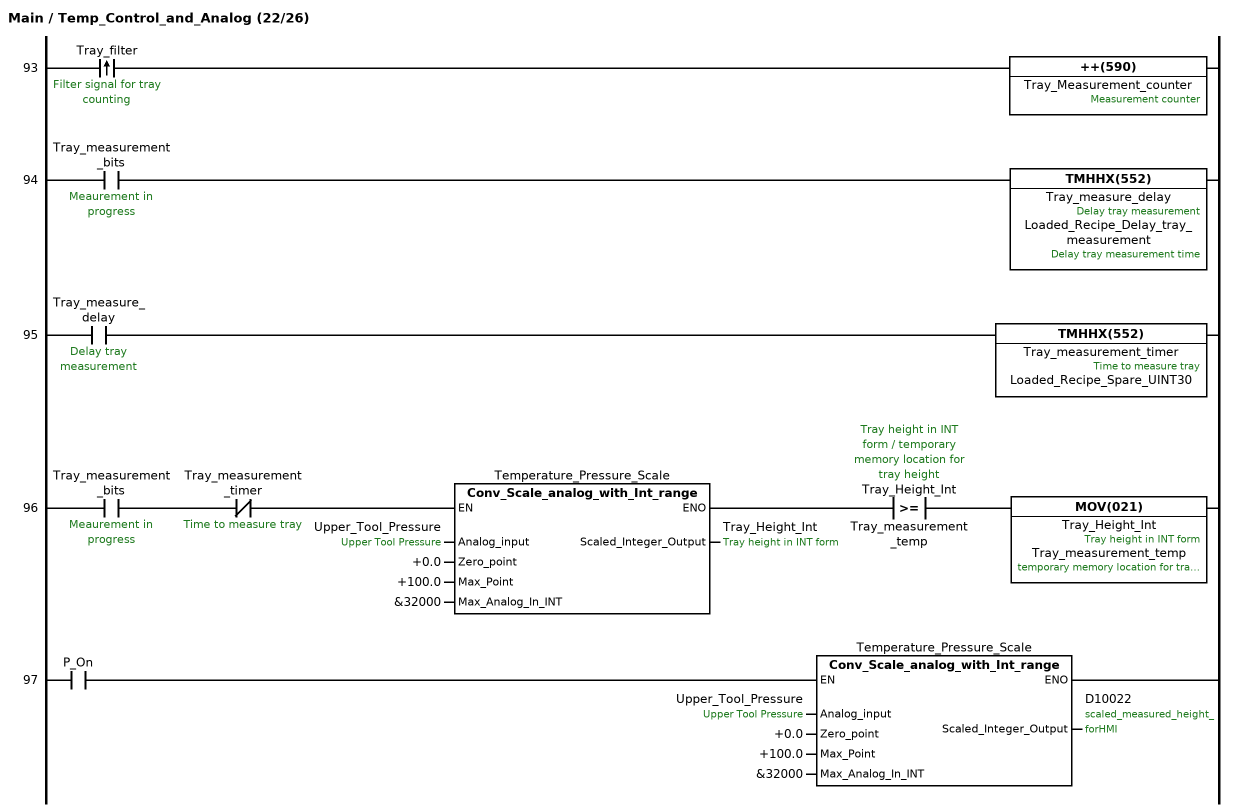
; [picture p120: Main / Temp_Control_and_Analog, rungs 93-97]
; rung 93
@LD Tray_filter  ; Filter signal for tray counting
++(590) Tray_Measurement_counter  ; Measurement counter
; rung 94
LD Tray_measurement_bits  ; Meaurement in progress
TMHHX(552) Tray_measure_delay Loaded_Recipe_Delay_tray_measurement  ; Delay tray measurement, Delay tray measurement time
; rung 95
LD Tray_measure_delay  ; Delay tray measurement
TMHHX(552) Tray_measurement_timer Loaded_Recipe_Spare_UINT30  ; Time to measure tray
; rung 96
LD Tray_measurement_bits  ; Meaurement in progress
ANDNOT Tray_measurement_timer  ; Time to measure tray
CALL Temperature_Pressure_Scale : Conv_Scale_analog_with_Int_range (Analog_input := Upper_Tool_Pressure, Zero_point := +0.0, Max_Point := +100.0, Max_Analog_In_INT := &32000, Scaled_Integer_Output => Tray_Height_Int)  ; Upper Tool Pressure, Tray height in INT form
AND>=(325) Tray_Height_Int Tray_measurement_temp  ; Tray height in INT form, temporary memory location for tray height
MOV(021) Tray_Height_Int Tray_measurement_temp  ; Tray height in INT form, temporary memory location for tray height
; rung 97
LD P_On
CALL Temperature_Pressure_Scale : Conv_Scale_analog_with_Int_range (Analog_input := Upper_Tool_Pressure, Zero_point := +0.0, Max_Point := +100.0, Max_Analog_In_INT := &32000, Scaled_Integer_Output => D10022)  ; Upper Tool Pressure, scaled_measured_height_forHMI

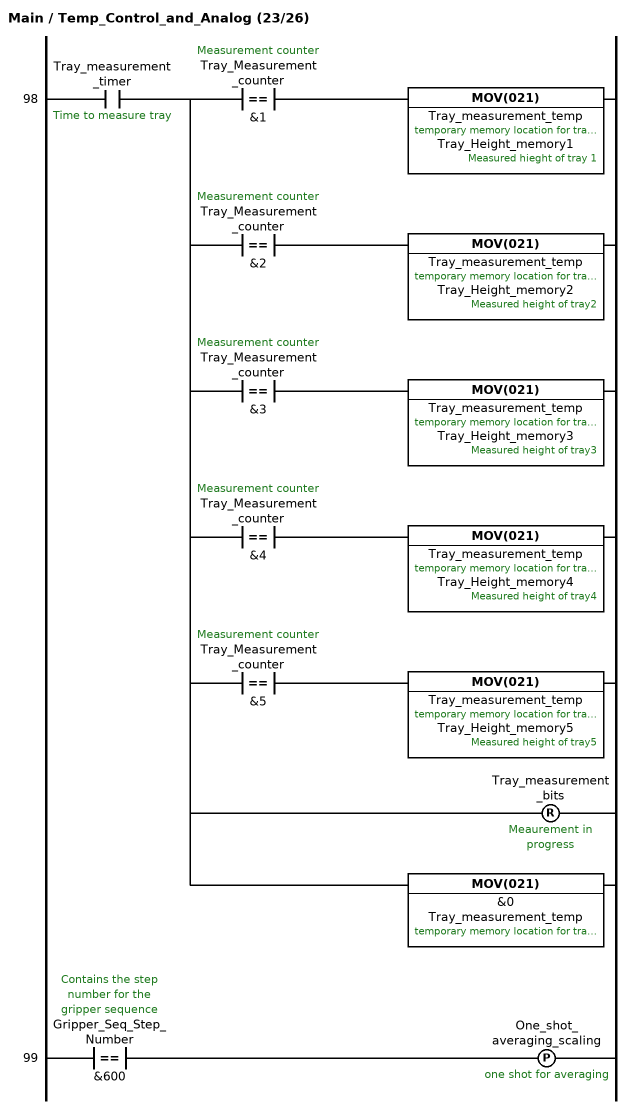
; rung 98
LD Tray_measurement_timer  ; Time to measure tray
OUT TR0
AND=(300) Tray_Measurement_counter &1  ; Measurement counter
MOV(021) Tray_measurement_temp Tray_Height_memory1  ; temporary memory location for tray height, Measured hieght of tray 1
LD TR0
AND=(300) Tray_Measurement_counter &2  ; Measurement counter
MOV(021) Tray_measurement_temp Tray_Height_memory2  ; temporary memory location for tray height, Measured height of tray2
LD TR0
AND=(300) Tray_Measurement_counter &3  ; Measurement counter
MOV(021) Tray_measurement_temp Tray_Height_memory3  ; temporary memory location for tray height, Measured height of tray3
LD TR0
AND=(300) Tray_Measurement_counter &4  ; Measurement counter
MOV(021) Tray_measurement_temp Tray_Height_memory4  ; temporary memory location for tray height, Measured height of tray4
LD TR0
AND=(300) Tray_Measurement_counter &5  ; Measurement counter
MOV(021) Tray_measurement_temp Tray_Height_memory5  ; temporary memory location for tray height, Measured height of tray5
LD TR0
RSET Tray_measurement_bits  ; Meaurement in progress
MOV(021) &0 Tray_measurement_temp  ; temporary memory location for tray height
; rung 99
LD=(300) Gripper_Seq_Step_Number &600  ; Contains the step number for the gripper sequence
DIFU(013) One_shot_averaging_scaling  ; one shot for averaging

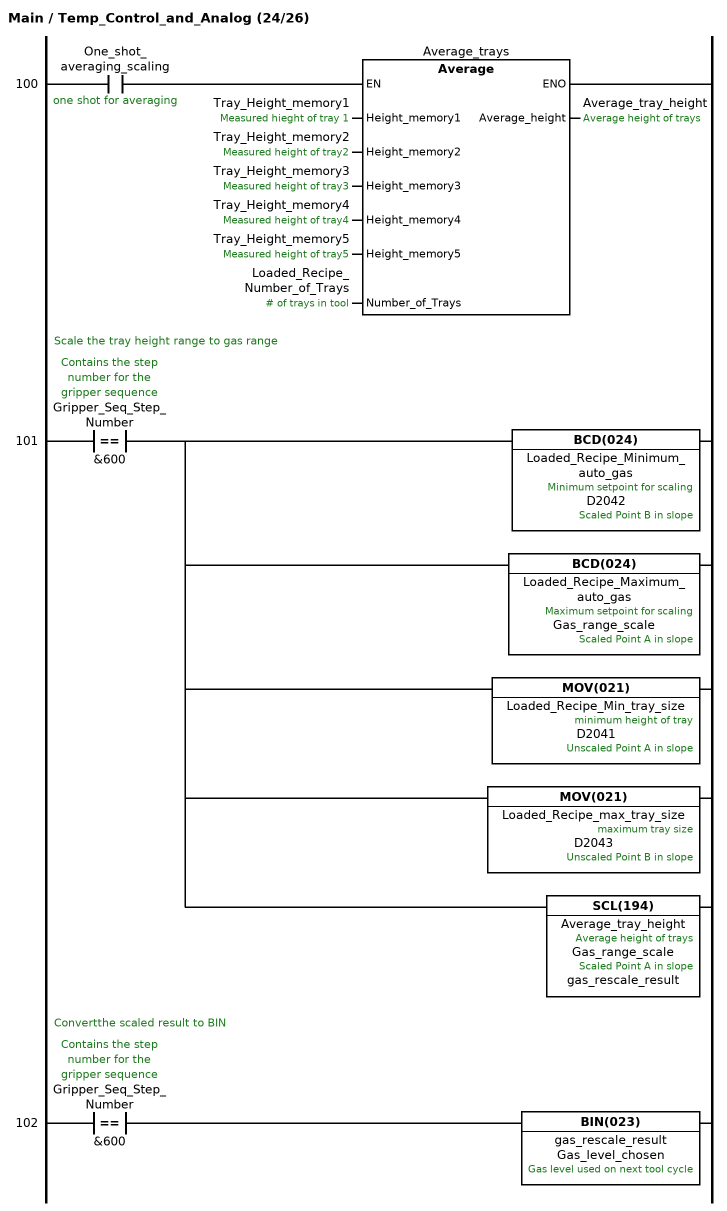
; rung 100
LD One_shot_averaging_scaling  ; one shot for averaging
CALL Average_trays : Average (Height_memory1 := Tray_Height_memory1, Height_memory2 := Tray_Height_memory2, Height_memory3 := Tray_Height_memory3, Height_memory4 := Tray_Height_memory4, Height_memory5 := Tray_Height_memory5, Number_of_Trays := Loaded_Recipe_Number_of_Trays, Average_height => Average_tray_height)  ; Measured hieght of tray 1, Measured height of tray2, Measured height of tray3, Measured height of tray4, Measured height of tray5, # of trays in tool, Average height of trays
; rung 101: Scale the tray height range to gas range
LD=(300) Gripper_Seq_Step_Number &600  ; Contains the step number for the gripper sequence
BCD(024) Loaded_Recipe_Minimum_auto_gas D2042  ; Minimum setpoint for scaling, Scaled Point B in slope
BCD(024) Loaded_Recipe_Maximum_auto_gas Gas_range_scale  ; Maximum setpoint for scaling, Scaled Point A in slope
MOV(021) Loaded_Recipe_Min_tray_size D2041  ; minimum height of tray, Unscaled Point A in slope
MOV(021) Loaded_Recipe_max_tray_size D2043  ; maximum tray size, Unscaled Point B in slope
SCL(194) Average_tray_height Gas_range_scale gas_rescale_result  ; Average height of trays, Scaled Point A in slope
; rung 102: Convertthe scaled result to BIN
LD=(300) Gripper_Seq_Step_Number &600  ; Contains the step number for the gripper sequence
BIN(023) gas_rescale_result Gas_level_chosen  ; Gas level used on next tool cycle

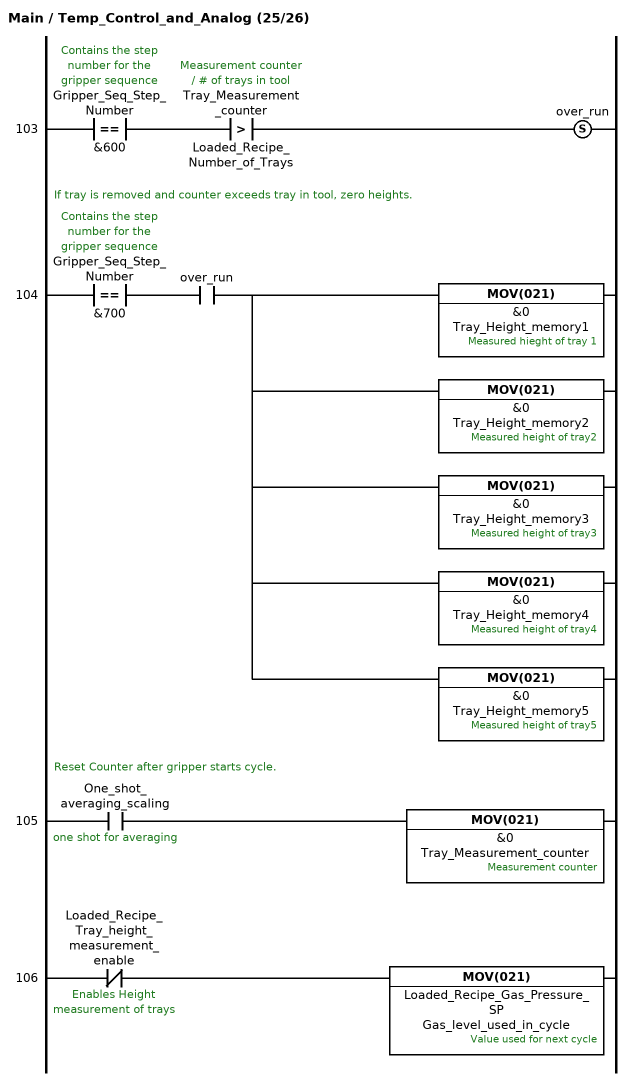
; rung 103
LD=(300) Gripper_Seq_Step_Number &600  ; Contains the step number for the gripper sequence
AND>(320) Tray_Measurement_counter Loaded_Recipe_Number_of_Trays  ; Measurement counter, # of trays in tool
SET over_run
; rung 104: If tray is removed and counter exceeds tray in tool, zero heights.
LD=(300) Gripper_Seq_Step_Number &700  ; Contains the step number for the gripper sequence
AND over_run
MOV(021) &0 Tray_Height_memory1  ; Measured hieght of tray 1
MOV(021) &0 Tray_Height_memory2  ; Measured height of tray2
MOV(021) &0 Tray_Height_memory3  ; Measured height of tray3
MOV(021) &0 Tray_Height_memory4  ; Measured height of tray4
MOV(021) &0 Tray_Height_memory5  ; Measured height of tray5
; rung 105: Reset Counter after gripper starts cycle.
LD One_shot_averaging_scaling  ; one shot for averaging
MOV(021) &0 Tray_Measurement_counter  ; Measurement counter
; rung 106
LDNOT Loaded_Recipe_Tray_height_measurement_enable  ; Enables Height measurement of trays
MOV(021) Loaded_Recipe_Gas_Pressure_SP Gas_level_used_in_cycle  ; Value used for next cycle

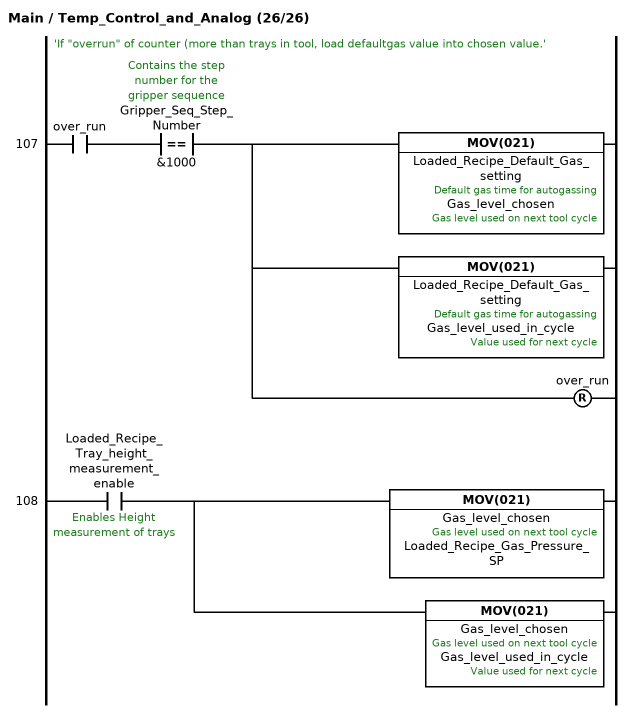
; rung 107: 'If "overrun" of counter (more than trays in tool, load defaultgas value into chosen value.'
LD over_run
AND=(300) Gripper_Seq_Step_Number &1000  ; Contains the step number for the gripper sequence
MOV(021) Loaded_Recipe_Default_Gas_setting Gas_level_chosen  ; Default gas time for autogassing, Gas level used on next tool cycle
MOV(021) Loaded_Recipe_Default_Gas_setting Gas_level_used_in_cycle  ; Default gas time for autogassing, Value used for next cycle
RSET over_run
; rung 108
LD Loaded_Recipe_Tray_height_measurement_enable  ; Enables Height measurement of trays
MOV(021) Gas_level_chosen Loaded_Recipe_Gas_Pressure_SP  ; Gas level used on next tool cycle
MOV(021) Gas_level_chosen Gas_level_used_in_cycle  ; Gas level used on next tool cycle, Value used for next cycle

### Section IOHandling

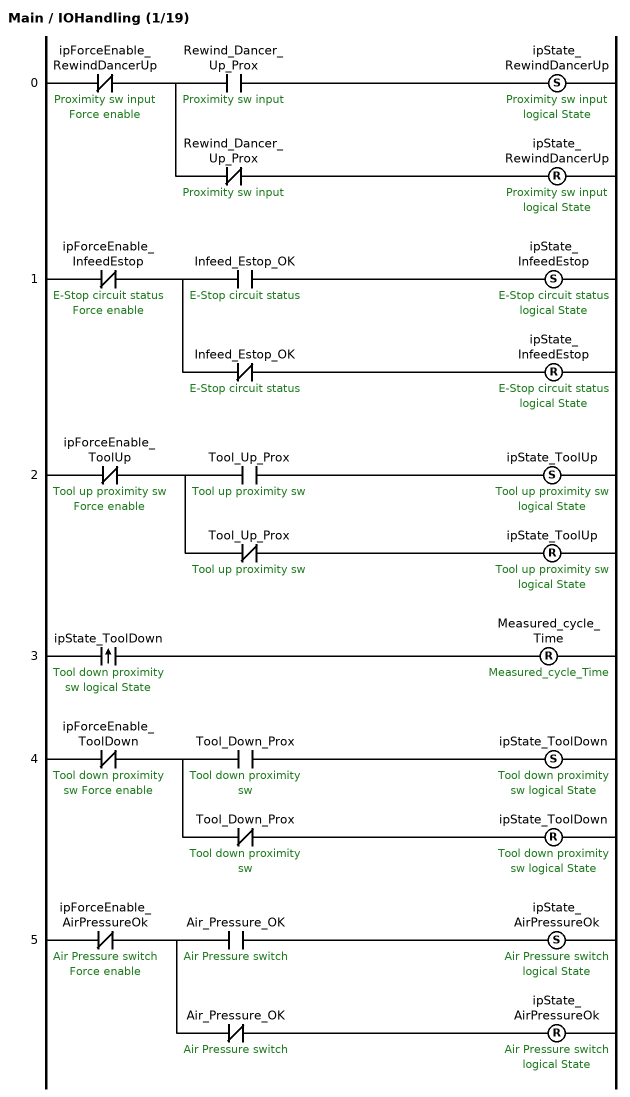
; rung 0
LDNOT ipForceEnable_RewindDancerUp  ; Proximity sw input Force enable
OUT TR0
AND Rewind_Dancer_Up_Prox  ; Proximity sw input
SET ipState_RewindDancerUp  ; Proximity sw input logical State
LD TR0
ANDNOT Rewind_Dancer_Up_Prox  ; Proximity sw input
RSET ipState_RewindDancerUp  ; Proximity sw input logical State
; rung 1
LDNOT ipForceEnable_InfeedEstop  ; E-Stop circuit status Force enable
OUT TR0
AND Infeed_Estop_OK  ; E-Stop circuit status
SET ipState_InfeedEstop  ; E-Stop circuit status logical State
LD TR0
ANDNOT Infeed_Estop_OK  ; E-Stop circuit status
RSET ipState_InfeedEstop  ; E-Stop circuit status logical State
; rung 2
LDNOT ipForceEnable_ToolUp  ; Tool up proximity sw Force enable
OUT TR0
AND Tool_Up_Prox  ; Tool up proximity sw
SET ipState_ToolUp  ; Tool up proximity sw logical State
LD TR0
ANDNOT Tool_Up_Prox  ; Tool up proximity sw
RSET ipState_ToolUp  ; Tool up proximity sw logical State
; rung 3
@LD ipState_ToolDown  ; Tool down proximity sw logical State
RSET Measured_cycle_Time  ; Measured_cycle_Time
; rung 4
LDNOT ipForceEnable_ToolDown  ; Tool down proximity sw Force enable
OUT TR0
AND Tool_Down_Prox  ; Tool down proximity sw
SET ipState_ToolDown  ; Tool down proximity sw logical State
LD TR0
ANDNOT Tool_Down_Prox  ; Tool down proximity sw
RSET ipState_ToolDown  ; Tool down proximity sw logical State
; rung 5
LDNOT ipForceEnable_AirPressureOk  ; Air Pressure switch Force enable
OUT TR0
AND Air_Pressure_OK  ; Air Pressure switch
SET ipState_AirPressureOk  ; Air Pressure switch logical State
LD TR0
ANDNOT Air_Pressure_OK  ; Air Pressure switch
RSET ipState_AirPressureOk  ; Air Pressure switch logical State

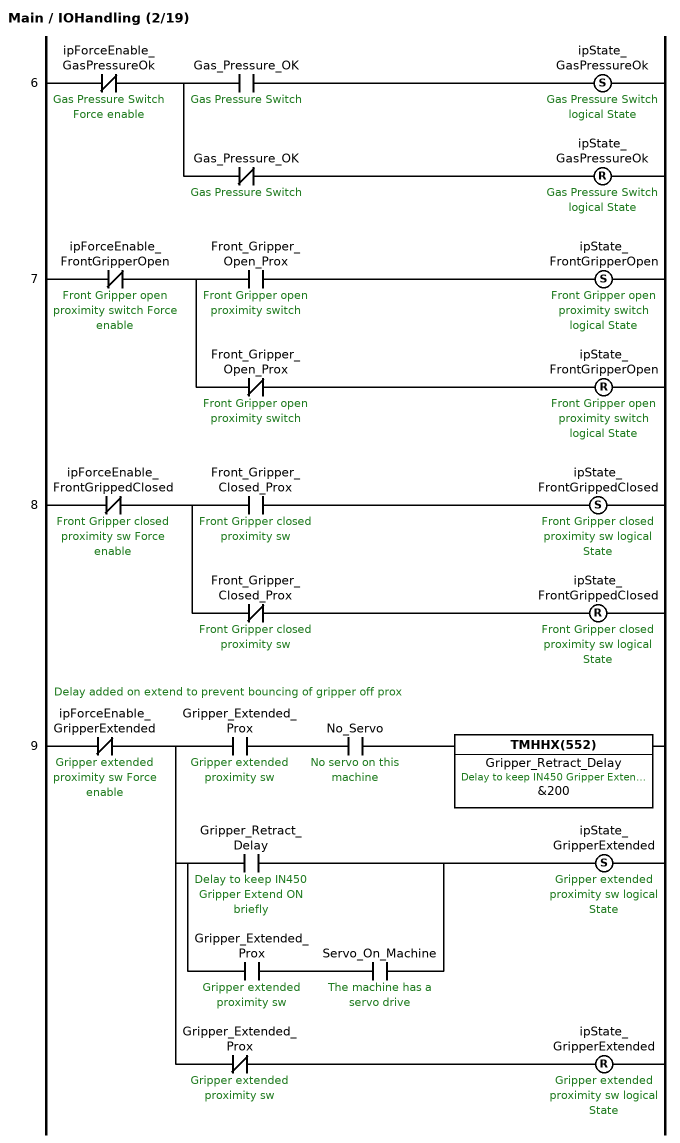
; rung 6
LDNOT ipForceEnable_GasPressureOk  ; Gas Pressure Switch Force enable
OUT TR0
AND Gas_Pressure_OK  ; Gas Pressure Switch
SET ipState_GasPressureOk  ; Gas Pressure Switch logical State
LD TR0
ANDNOT Gas_Pressure_OK  ; Gas Pressure Switch
RSET ipState_GasPressureOk  ; Gas Pressure Switch logical State
; rung 7
LDNOT ipForceEnable_FrontGripperOpen  ; Front Gripper open proximity switch Force enable
OUT TR0
AND Front_Gripper_Open_Prox  ; Front Gripper open proximity switch
SET ipState_FrontGripperOpen  ; Front Gripper open proximity switch logical State
LD TR0
ANDNOT Front_Gripper_Open_Prox  ; Front Gripper open proximity switch
RSET ipState_FrontGripperOpen  ; Front Gripper open proximity switch logical State
; rung 8
LDNOT ipForceEnable_FrontGrippedClosed  ; Front Gripper closed proximity sw Force enable
OUT TR0
AND Front_Gripper_Closed_Prox  ; Front Gripper closed proximity sw
SET ipState_FrontGrippedClosed  ; Front Gripper closed proximity sw logical State
LD TR0
ANDNOT Front_Gripper_Closed_Prox  ; Front Gripper closed proximity sw
RSET ipState_FrontGrippedClosed  ; Front Gripper closed proximity sw logical State
; rung 9: Delay added on extend to prevent bouncing of gripper off prox
LDNOT ipForceEnable_GripperExtended  ; Gripper extended proximity sw Force enable
OUT TR0
AND Gripper_Extended_Prox  ; Gripper extended proximity sw
AND No_Servo  ; No servo on this machine
TMHHX(552) Gripper_Retract_Delay &200  ; Delay to keep IN450 Gripper Extend ON briefly
LD TR0
LD Gripper_Retract_Delay  ; Delay to keep IN450 Gripper Extend ON briefly
LD Gripper_Extended_Prox  ; Gripper extended proximity sw
AND Servo_On_Machine  ; The machine has a servo drive
ORLD
ANDLD
SET ipState_GripperExtended  ; Gripper extended proximity sw logical State
LD TR0
ANDNOT Gripper_Extended_Prox  ; Gripper extended proximity sw
RSET ipState_GripperExtended  ; Gripper extended proximity sw logical State

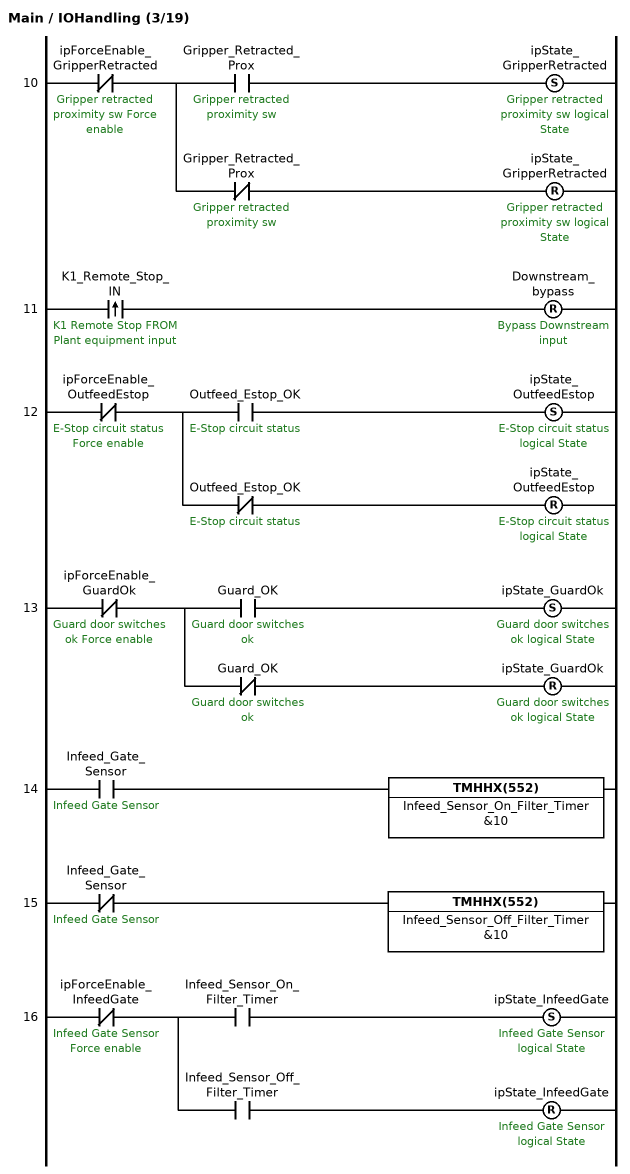
; rung 10
LDNOT ipForceEnable_GripperRetracted  ; Gripper retracted proximity sw Force enable
OUT TR0
AND Gripper_Retracted_Prox  ; Gripper retracted proximity sw
SET ipState_GripperRetracted  ; Gripper retracted proximity sw logical State
LD TR0
ANDNOT Gripper_Retracted_Prox  ; Gripper retracted proximity sw
RSET ipState_GripperRetracted  ; Gripper retracted proximity sw logical State
; rung 11
@LD K1_Remote_Stop_IN  ; K1 Remote Stop FROM Plant equipment input
RSET Downstream_bypass  ; Bypass Downstream input
; rung 12
LDNOT ipForceEnable_OutfeedEstop  ; E-Stop circuit status Force enable
OUT TR0
AND Outfeed_Estop_OK  ; E-Stop circuit status
SET ipState_OutfeedEstop  ; E-Stop circuit status logical State
LD TR0
ANDNOT Outfeed_Estop_OK  ; E-Stop circuit status
RSET ipState_OutfeedEstop  ; E-Stop circuit status logical State
; rung 13
LDNOT ipForceEnable_GuardOk  ; Guard door switches ok Force enable
OUT TR0
AND Guard_OK  ; Guard door switches ok
SET ipState_GuardOk  ; Guard door switches ok logical State
LD TR0
ANDNOT Guard_OK  ; Guard door switches ok
RSET ipState_GuardOk  ; Guard door switches ok logical State
; rung 14
LD Infeed_Gate_Sensor  ; Infeed Gate Sensor
TMHHX(552) Infeed_Sensor_On_Filter_Timer &10
; rung 15
LDNOT Infeed_Gate_Sensor  ; Infeed Gate Sensor
TMHHX(552) Infeed_Sensor_Off_Filter_Timer &10
; rung 16
LDNOT ipForceEnable_InfeedGate  ; Infeed Gate Sensor Force enable
OUT TR0
AND Infeed_Sensor_On_Filter_Timer
SET ipState_InfeedGate  ; Infeed Gate Sensor logical State
LD TR0
AND Infeed_Sensor_Off_Filter_Timer
RSET ipState_InfeedGate  ; Infeed Gate Sensor logical State

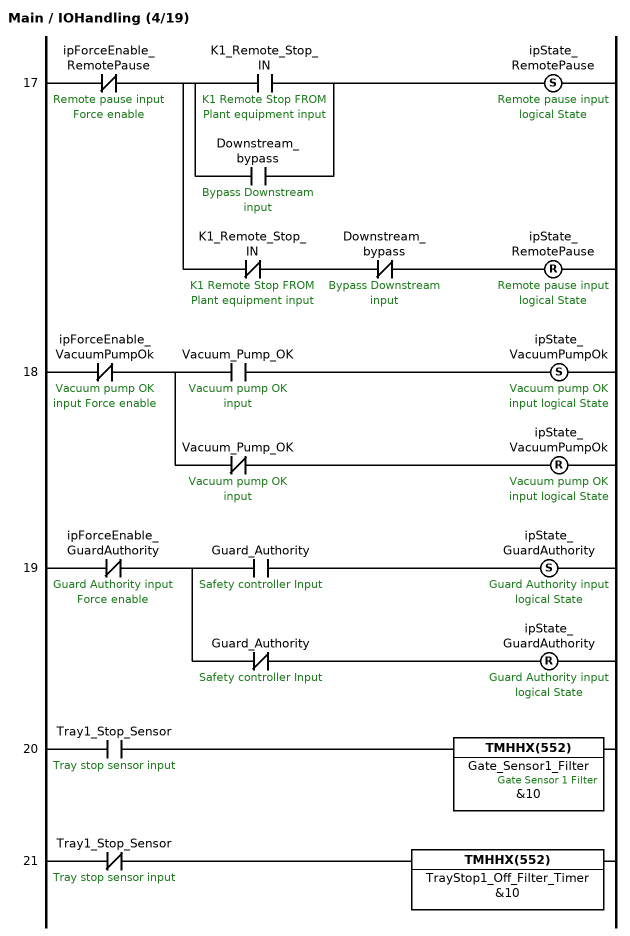
; rung 17
LDNOT ipForceEnable_RemotePause  ; Remote pause input Force enable
OUT TR0
LD K1_Remote_Stop_IN  ; K1 Remote Stop FROM Plant equipment input
OR Downstream_bypass  ; Bypass Downstream input
ANDLD
SET ipState_RemotePause  ; Remote pause input logical State
LD TR0
ANDNOT K1_Remote_Stop_IN  ; K1 Remote Stop FROM Plant equipment input
ANDNOT Downstream_bypass  ; Bypass Downstream input
RSET ipState_RemotePause  ; Remote pause input logical State
; rung 18
LDNOT ipForceEnable_VacuumPumpOk  ; Vacuum pump OK input Force enable
OUT TR0
AND Vacuum_Pump_OK  ; Vacuum pump OK input
SET ipState_VacuumPumpOk  ; Vacuum pump OK input logical State
LD TR0
ANDNOT Vacuum_Pump_OK  ; Vacuum pump OK input
RSET ipState_VacuumPumpOk  ; Vacuum pump OK input logical State
; rung 19
LDNOT ipForceEnable_GuardAuthority  ; Guard Authority input Force enable
OUT TR0
AND Guard_Authority  ; Safety controller Input
SET ipState_GuardAuthority  ; Guard Authority input logical State
LD TR0
ANDNOT Guard_Authority  ; Safety controller Input
RSET ipState_GuardAuthority  ; Guard Authority input logical State
; rung 20
LD Tray1_Stop_Sensor  ; Tray stop sensor input
TMHHX(552) Gate_Sensor1_Filter &10  ; Gate Sensor 1 Filter
; rung 21
LDNOT Tray1_Stop_Sensor  ; Tray stop sensor input
TMHHX(552) TrayStop1_Off_Filter_Timer &10

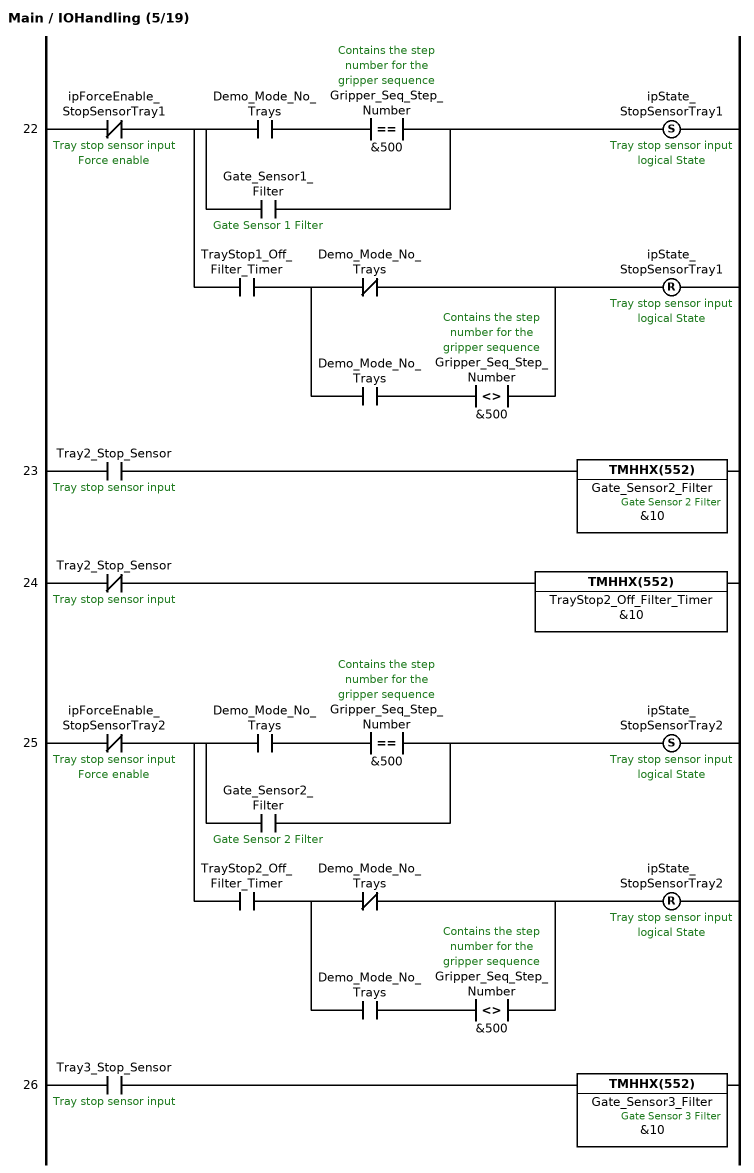
; rung 22
LDNOT ipForceEnable_StopSensorTray1  ; Tray stop sensor input Force enable
OUT TR0
LD Demo_Mode_No_Trays
AND=(300) Gripper_Seq_Step_Number &500  ; Contains the step number for the gripper sequence
OR Gate_Sensor1_Filter  ; Gate Sensor 1 Filter
ANDLD
SET ipState_StopSensorTray1  ; Tray stop sensor input logical State
LD TR0
AND TrayStop1_Off_Filter_Timer
LDNOT Demo_Mode_No_Trays
LD Demo_Mode_No_Trays
AND<>(305) Gripper_Seq_Step_Number &500  ; Contains the step number for the gripper sequence
ORLD
ANDLD
RSET ipState_StopSensorTray1  ; Tray stop sensor input logical State
; rung 23
LD Tray2_Stop_Sensor  ; Tray stop sensor input
TMHHX(552) Gate_Sensor2_Filter &10  ; Gate Sensor 2 Filter
; rung 24
LDNOT Tray2_Stop_Sensor  ; Tray stop sensor input
TMHHX(552) TrayStop2_Off_Filter_Timer &10
; rung 25
LDNOT ipForceEnable_StopSensorTray2  ; Tray stop sensor input Force enable
OUT TR0
LD Demo_Mode_No_Trays
AND=(300) Gripper_Seq_Step_Number &500  ; Contains the step number for the gripper sequence
OR Gate_Sensor2_Filter  ; Gate Sensor 2 Filter
ANDLD
SET ipState_StopSensorTray2  ; Tray stop sensor input logical State
LD TR0
AND TrayStop2_Off_Filter_Timer
LDNOT Demo_Mode_No_Trays
LD Demo_Mode_No_Trays
AND<>(305) Gripper_Seq_Step_Number &500  ; Contains the step number for the gripper sequence
ORLD
ANDLD
RSET ipState_StopSensorTray2  ; Tray stop sensor input logical State
; rung 26
LD Tray3_Stop_Sensor  ; Tray stop sensor input
TMHHX(552) Gate_Sensor3_Filter &10  ; Gate Sensor 3 Filter

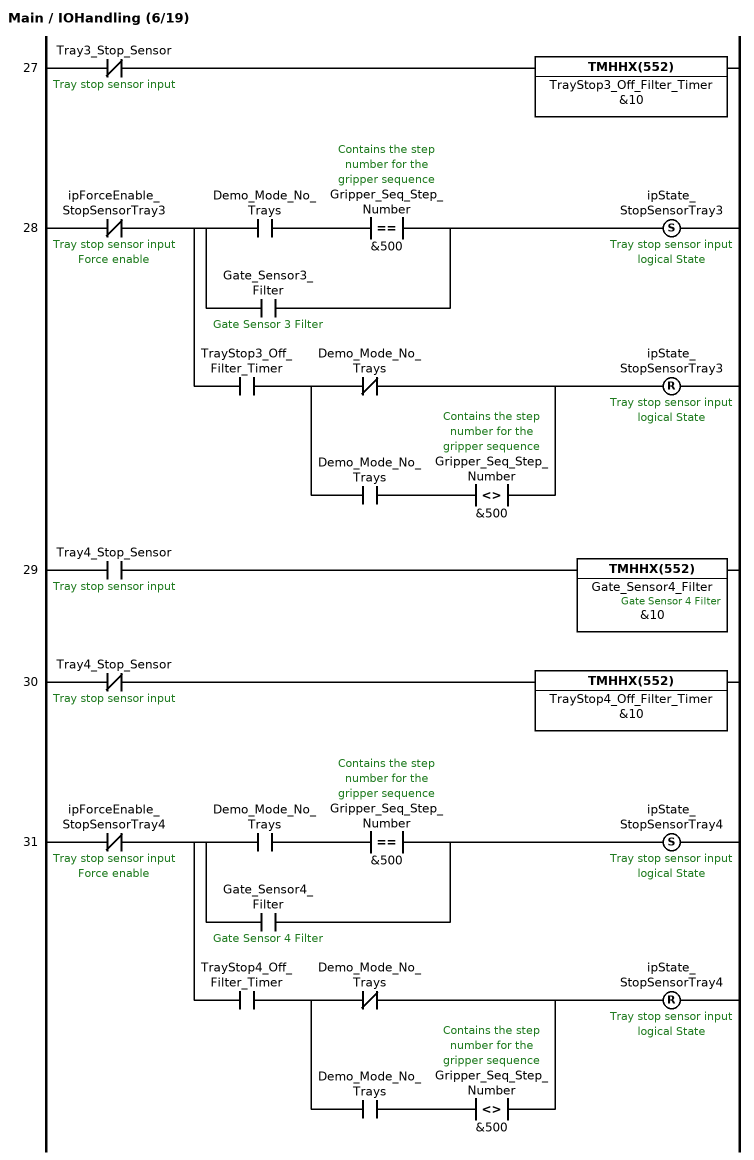
; rung 27
LDNOT Tray3_Stop_Sensor  ; Tray stop sensor input
TMHHX(552) TrayStop3_Off_Filter_Timer &10
; rung 28
LDNOT ipForceEnable_StopSensorTray3  ; Tray stop sensor input Force enable
OUT TR0
LD Demo_Mode_No_Trays
AND=(300) Gripper_Seq_Step_Number &500  ; Contains the step number for the gripper sequence
OR Gate_Sensor3_Filter  ; Gate Sensor 3 Filter
ANDLD
SET ipState_StopSensorTray3  ; Tray stop sensor input logical State
LD TR0
AND TrayStop3_Off_Filter_Timer
LDNOT Demo_Mode_No_Trays
LD Demo_Mode_No_Trays
AND<>(305) Gripper_Seq_Step_Number &500  ; Contains the step number for the gripper sequence
ORLD
ANDLD
RSET ipState_StopSensorTray3  ; Tray stop sensor input logical State
; rung 29
LD Tray4_Stop_Sensor  ; Tray stop sensor input
TMHHX(552) Gate_Sensor4_Filter &10  ; Gate Sensor 4 Filter
; rung 30
LDNOT Tray4_Stop_Sensor  ; Tray stop sensor input
TMHHX(552) TrayStop4_Off_Filter_Timer &10
; rung 31
LDNOT ipForceEnable_StopSensorTray4  ; Tray stop sensor input Force enable
OUT TR0
LD Demo_Mode_No_Trays
AND=(300) Gripper_Seq_Step_Number &500  ; Contains the step number for the gripper sequence
OR Gate_Sensor4_Filter  ; Gate Sensor 4 Filter
ANDLD
SET ipState_StopSensorTray4  ; Tray stop sensor input logical State
LD TR0
AND TrayStop4_Off_Filter_Timer
LDNOT Demo_Mode_No_Trays
LD Demo_Mode_No_Trays
AND<>(305) Gripper_Seq_Step_Number &500  ; Contains the step number for the gripper sequence
ORLD
ANDLD
RSET ipState_StopSensorTray4  ; Tray stop sensor input logical State

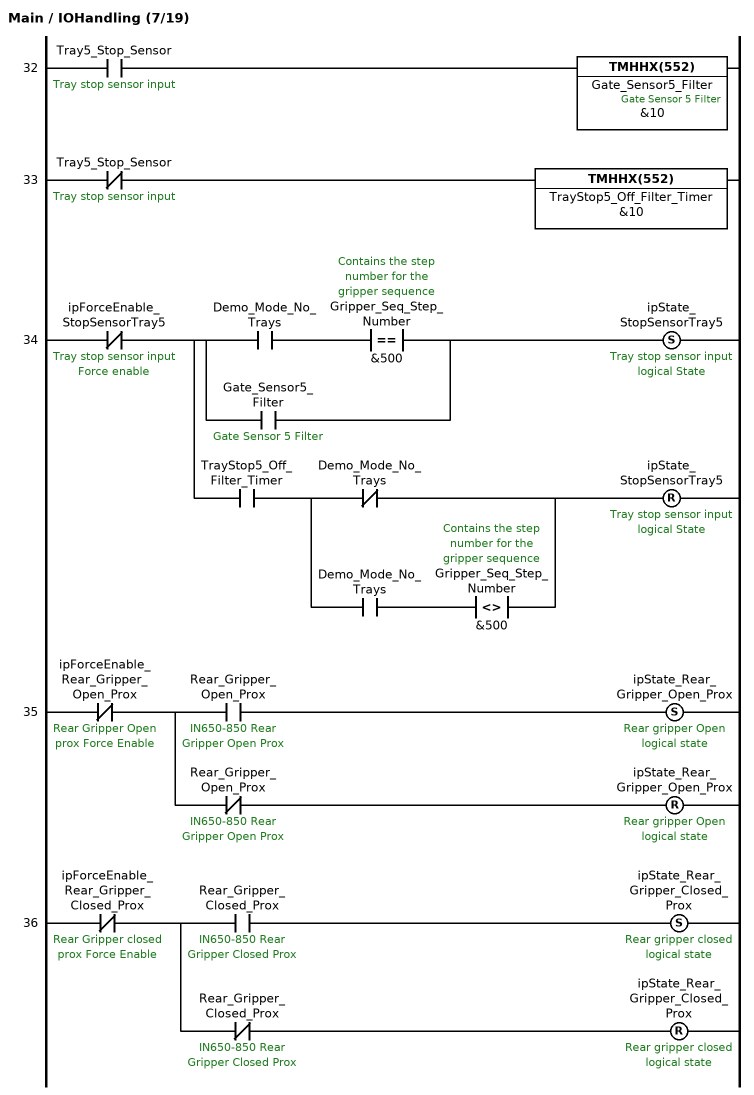
; rung 32
LD Tray5_Stop_Sensor  ; Tray stop sensor input
TMHHX(552) Gate_Sensor5_Filter &10  ; Gate Sensor 5 Filter
; rung 33
LDNOT Tray5_Stop_Sensor  ; Tray stop sensor input
TMHHX(552) TrayStop5_Off_Filter_Timer &10
; rung 34
LDNOT ipForceEnable_StopSensorTray5  ; Tray stop sensor input Force enable
OUT TR0
LD Demo_Mode_No_Trays
AND=(300) Gripper_Seq_Step_Number &500  ; Contains the step number for the gripper sequence
OR Gate_Sensor5_Filter  ; Gate Sensor 5 Filter
ANDLD
SET ipState_StopSensorTray5  ; Tray stop sensor input logical State
LD TR0
AND TrayStop5_Off_Filter_Timer
LDNOT Demo_Mode_No_Trays
LD Demo_Mode_No_Trays
AND<>(305) Gripper_Seq_Step_Number &500  ; Contains the step number for the gripper sequence
ORLD
ANDLD
RSET ipState_StopSensorTray5  ; Tray stop sensor input logical State
; rung 35
LDNOT ipForceEnable_Rear_Gripper_Open_Prox  ; Rear Gripper Open prox Force Enable
OUT TR0
AND Rear_Gripper_Open_Prox  ; IN650-850 Rear Gripper Open Prox
SET ipState_Rear_Gripper_Open_Prox  ; Rear gripper Open logical state
LD TR0
ANDNOT Rear_Gripper_Open_Prox  ; IN650-850 Rear Gripper Open Prox
RSET ipState_Rear_Gripper_Open_Prox  ; Rear gripper Open logical state
; rung 36
LDNOT ipForceEnable_Rear_Gripper_Closed_Prox  ; Rear Gripper closed prox Force Enable
OUT TR0
AND Rear_Gripper_Closed_Prox  ; IN650-850 Rear Gripper Closed Prox
SET ipState_Rear_Gripper_Closed_Prox  ; Rear gripper closed logical state
LD TR0
ANDNOT Rear_Gripper_Closed_Prox  ; IN650-850 Rear Gripper Closed Prox
RSET ipState_Rear_Gripper_Closed_Prox  ; Rear gripper closed logical state

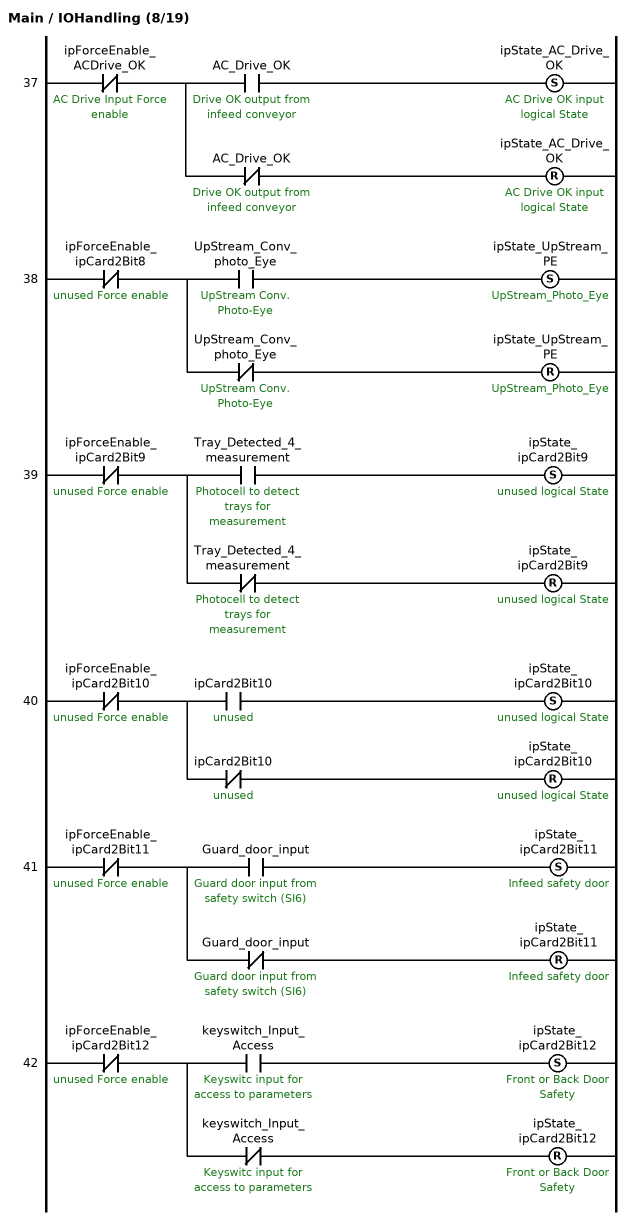
; rung 37
LDNOT ipForceEnable_ACDrive_OK  ; AC Drive Input Force enable
OUT TR0
AND AC_Drive_OK  ; Drive OK output from infeed conveyor
SET ipState_AC_Drive_OK  ; AC Drive OK input logical State
LD TR0
ANDNOT AC_Drive_OK  ; Drive OK output from infeed conveyor
RSET ipState_AC_Drive_OK  ; AC Drive OK input logical State
; rung 38
LDNOT ipForceEnable_ipCard2Bit8  ; unused Force enable
OUT TR0
AND UpStream_Conv_photo_Eye  ; UpStream Conv. Photo-Eye
SET ipState_UpStream_PE  ; UpStream_Photo_Eye
LD TR0
ANDNOT UpStream_Conv_photo_Eye  ; UpStream Conv. Photo-Eye
RSET ipState_UpStream_PE  ; UpStream_Photo_Eye
; rung 39
LDNOT ipForceEnable_ipCard2Bit9  ; unused Force enable
OUT TR0
AND Tray_Detected_4_measurement  ; Photocell to detect trays for measurement
SET ipState_ipCard2Bit9  ; unused logical State
LD TR0
ANDNOT Tray_Detected_4_measurement  ; Photocell to detect trays for measurement
RSET ipState_ipCard2Bit9  ; unused logical State
; rung 40
LDNOT ipForceEnable_ipCard2Bit10  ; unused Force enable
OUT TR0
AND ipCard2Bit10  ; unused
SET ipState_ipCard2Bit10  ; unused logical State
LD TR0
ANDNOT ipCard2Bit10  ; unused
RSET ipState_ipCard2Bit10  ; unused logical State
; rung 41
LDNOT ipForceEnable_ipCard2Bit11  ; unused Force enable
OUT TR0
AND Guard_door_input  ; Guard door input from safety switch (SI6)
SET ipState_ipCard2Bit11  ; Infeed safety door
LD TR0
ANDNOT Guard_door_input  ; Guard door input from safety switch (SI6)
RSET ipState_ipCard2Bit11  ; Infeed safety door
; rung 42
LDNOT ipForceEnable_ipCard2Bit12  ; unused Force enable
OUT TR0
AND keyswitch_Input_Access  ; Keyswitc input for access to parameters
SET ipState_ipCard2Bit12  ; Front or Back Door Safety
LD TR0
ANDNOT keyswitch_Input_Access  ; Keyswitc input for access to parameters
RSET ipState_ipCard2Bit12  ; Front or Back Door Safety

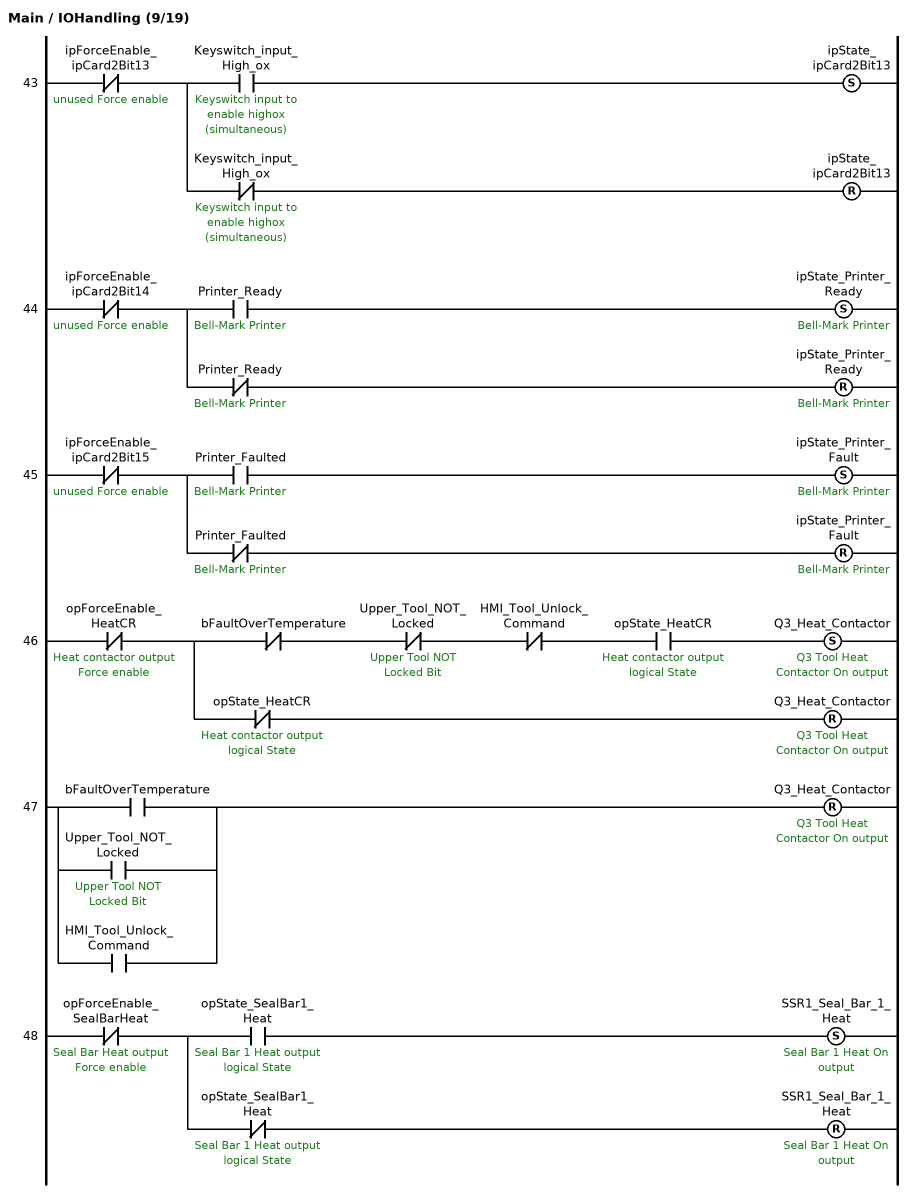
; rung 43
LDNOT ipForceEnable_ipCard2Bit13  ; unused Force enable
OUT TR0
AND Keyswitch_input_High_ox  ; Keyswitch input to enable highox (simultaneous)
SET ipState_ipCard2Bit13
LD TR0
ANDNOT Keyswitch_input_High_ox  ; Keyswitch input to enable highox (simultaneous)
RSET ipState_ipCard2Bit13
; rung 44
LDNOT ipForceEnable_ipCard2Bit14  ; unused Force enable
OUT TR0
AND Printer_Ready  ; Bell-Mark Printer
SET ipState_Printer_Ready  ; Bell-Mark Printer
LD TR0
ANDNOT Printer_Ready  ; Bell-Mark Printer
RSET ipState_Printer_Ready  ; Bell-Mark Printer
; rung 45
LDNOT ipForceEnable_ipCard2Bit15  ; unused Force enable
OUT TR0
AND Printer_Faulted  ; Bell-Mark Printer
SET ipState_Printer_Fault  ; Bell-Mark Printer
LD TR0
ANDNOT Printer_Faulted  ; Bell-Mark Printer
RSET ipState_Printer_Fault  ; Bell-Mark Printer
; rung 46
LDNOT opForceEnable_HeatCR  ; Heat contactor output Force enable
OUT TR0
ANDNOT bFaultOverTemperature
ANDNOT Upper_Tool_NOT_Locked  ; Upper Tool NOT Locked Bit
ANDNOT HMI_Tool_Unlock_Command
AND opState_HeatCR  ; Heat contactor output logical State
SET Q3_Heat_Contactor  ; Q3 Tool Heat Contactor On output
LD TR0
ANDNOT opState_HeatCR  ; Heat contactor output logical State
RSET Q3_Heat_Contactor  ; Q3 Tool Heat Contactor On output
; rung 47
LD bFaultOverTemperature
OR Upper_Tool_NOT_Locked  ; Upper Tool NOT Locked Bit
OR HMI_Tool_Unlock_Command
RSET Q3_Heat_Contactor  ; Q3 Tool Heat Contactor On output
; rung 48
LDNOT opForceEnable_SealBarHeat  ; Seal Bar Heat output Force enable
OUT TR0
AND opState_SealBar1_Heat  ; Seal Bar 1 Heat output logical State
SET SSR1_Seal_Bar_1_Heat  ; Seal Bar 1 Heat On output
LD TR0
ANDNOT opState_SealBar1_Heat  ; Seal Bar 1 Heat output logical State
RSET SSR1_Seal_Bar_1_Heat  ; Seal Bar 1 Heat On output

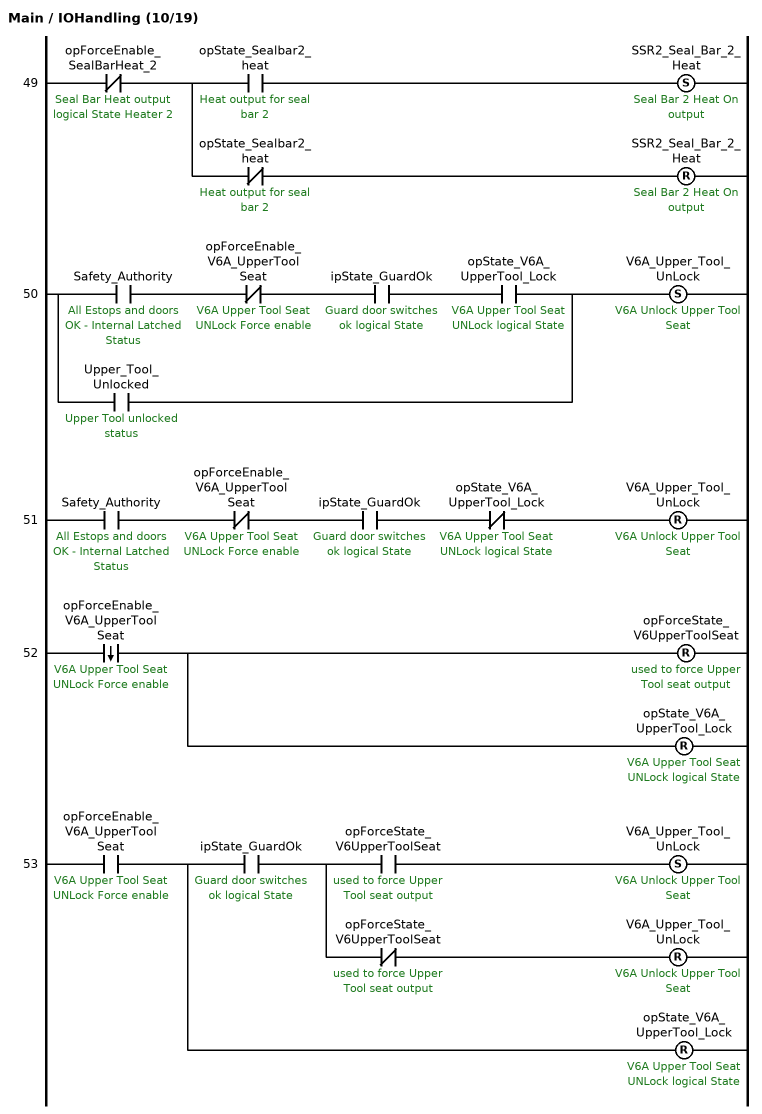
; rung 49
LDNOT opForceEnable_SealBarHeat_2  ; Seal Bar Heat output logical State Heater 2
OUT TR0
AND opState_Sealbar2_heat  ; Heat output for seal bar 2
SET SSR2_Seal_Bar_2_Heat  ; Seal Bar 2 Heat On output
LD TR0
ANDNOT opState_Sealbar2_heat  ; Heat output for seal bar 2
RSET SSR2_Seal_Bar_2_Heat  ; Seal Bar 2 Heat On output
; rung 50
LD Safety_Authority  ; All Estops and doors OK - Internal Latched Status
ANDNOT opForceEnable_V6A_UpperToolSeat  ; V6A Upper Tool Seat UNLock Force enable
AND ipState_GuardOk  ; Guard door switches ok logical State
AND opState_V6A_UpperTool_Lock  ; V6A Upper Tool Seat UNLock logical State
OR Upper_Tool_Unlocked  ; Upper Tool unlocked status
SET V6A_Upper_Tool_UnLock  ; V6A Unlock Upper Tool Seat
; rung 51
LD Safety_Authority  ; All Estops and doors OK - Internal Latched Status
ANDNOT opForceEnable_V6A_UpperToolSeat  ; V6A Upper Tool Seat UNLock Force enable
AND ipState_GuardOk  ; Guard door switches ok logical State
ANDNOT opState_V6A_UpperTool_Lock  ; V6A Upper Tool Seat UNLock logical State
RSET V6A_Upper_Tool_UnLock  ; V6A Unlock Upper Tool Seat
; rung 52
%LD opForceEnable_V6A_UpperToolSeat  ; V6A Upper Tool Seat UNLock Force enable
RSET opForceState_V6UpperToolSeat  ; used to force Upper Tool seat output
RSET opState_V6A_UpperTool_Lock  ; V6A Upper Tool Seat UNLock logical State
; rung 53
LD opForceEnable_V6A_UpperToolSeat  ; V6A Upper Tool Seat UNLock Force enable
OUT TR0
AND ipState_GuardOk  ; Guard door switches ok logical State
OUT TR1
AND opForceState_V6UpperToolSeat  ; used to force Upper Tool seat output
SET V6A_Upper_Tool_UnLock  ; V6A Unlock Upper Tool Seat
LD TR1
ANDNOT opForceState_V6UpperToolSeat  ; used to force Upper Tool seat output
RSET V6A_Upper_Tool_UnLock  ; V6A Unlock Upper Tool Seat
LD TR0
RSET opState_V6A_UpperTool_Lock  ; V6A Upper Tool Seat UNLock logical State

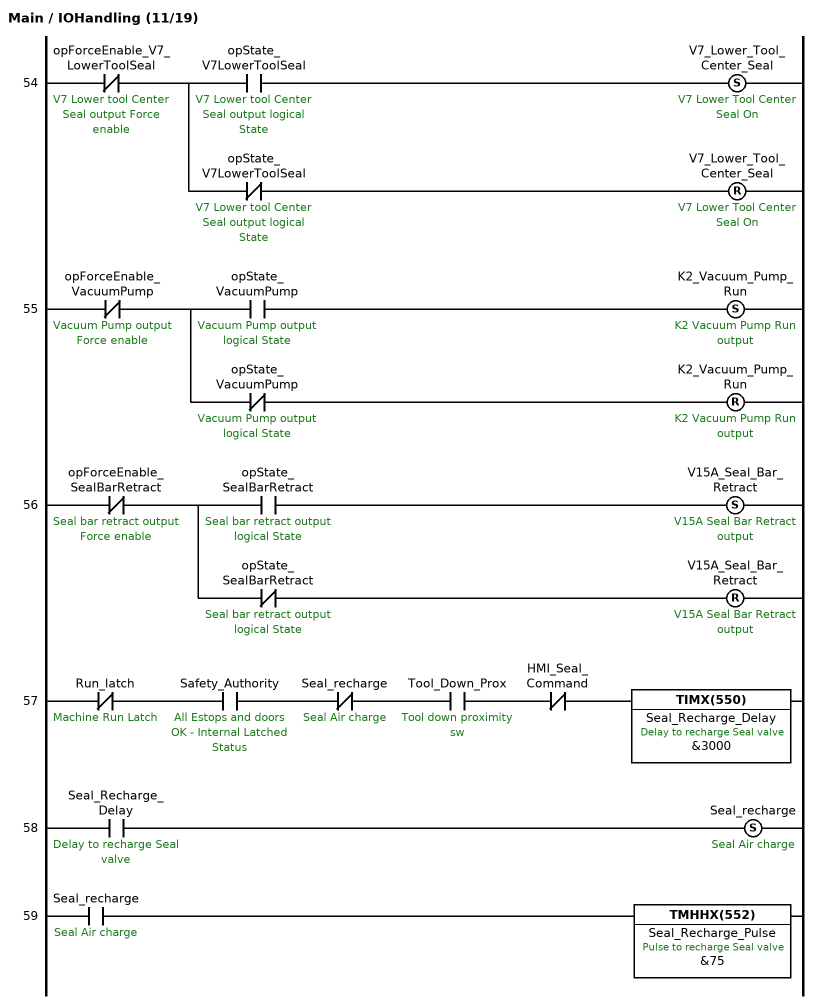
; rung 54
LDNOT opForceEnable_V7_LowerToolSeal  ; V7 Lower tool Center Seal output Force enable
OUT TR0
AND opState_V7LowerToolSeal  ; V7 Lower tool Center Seal output logical State
SET V7_Lower_Tool_Center_Seal  ; V7 Lower Tool Center Seal On
LD TR0
ANDNOT opState_V7LowerToolSeal  ; V7 Lower tool Center Seal output logical State
RSET V7_Lower_Tool_Center_Seal  ; V7 Lower Tool Center Seal On
; rung 55
LDNOT opForceEnable_VacuumPump  ; Vacuum Pump output Force enable
OUT TR0
AND opState_VacuumPump  ; Vacuum Pump output logical State
SET K2_Vacuum_Pump_Run  ; K2 Vacuum Pump Run output
LD TR0
ANDNOT opState_VacuumPump  ; Vacuum Pump output logical State
RSET K2_Vacuum_Pump_Run  ; K2 Vacuum Pump Run output
; rung 56
LDNOT opForceEnable_SealBarRetract  ; Seal bar retract output Force enable
OUT TR0
AND opState_SealBarRetract  ; Seal bar retract output logical State
SET V15A_Seal_Bar_Retract  ; V15A Seal Bar Retract output
LD TR0
ANDNOT opState_SealBarRetract  ; Seal bar retract output logical State
RSET V15A_Seal_Bar_Retract  ; V15A Seal Bar Retract output
; rung 57
LDNOT Run_latch  ; Machine Run Latch
AND Safety_Authority  ; All Estops and doors OK - Internal Latched Status
ANDNOT Seal_recharge  ; Seal Air charge
AND Tool_Down_Prox  ; Tool down proximity sw
ANDNOT HMI_Seal_Command
TIMX(550) Seal_Recharge_Delay &3000  ; Delay to recharge Seal valve
; rung 58
LD Seal_Recharge_Delay  ; Delay to recharge Seal valve
SET Seal_recharge  ; Seal Air charge
; rung 59
LD Seal_recharge  ; Seal Air charge
TMHHX(552) Seal_Recharge_Pulse &75  ; Pulse to recharge Seal valve

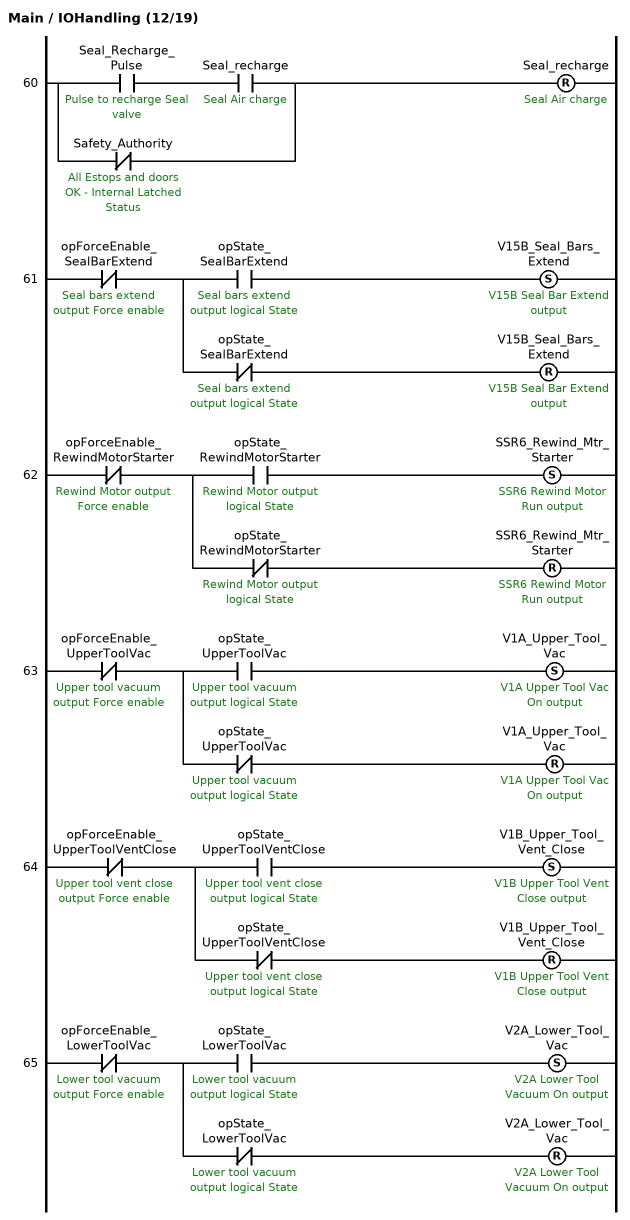
; rung 60
LD Seal_Recharge_Pulse  ; Pulse to recharge Seal valve
AND Seal_recharge  ; Seal Air charge
ORNOT Safety_Authority  ; All Estops and doors OK - Internal Latched Status
RSET Seal_recharge  ; Seal Air charge
; rung 61
LDNOT opForceEnable_SealBarExtend  ; Seal bars extend output Force enable
OUT TR0
AND opState_SealBarExtend  ; Seal bars extend output logical State
SET V15B_Seal_Bars_Extend  ; V15B Seal Bar Extend output
LD TR0
ANDNOT opState_SealBarExtend  ; Seal bars extend output logical State
RSET V15B_Seal_Bars_Extend  ; V15B Seal Bar Extend output
; rung 62
LDNOT opForceEnable_RewindMotorStarter  ; Rewind Motor output Force enable
OUT TR0
AND opState_RewindMotorStarter  ; Rewind Motor output logical State
SET SSR6_Rewind_Mtr_Starter  ; SSR6 Rewind Motor Run output
LD TR0
ANDNOT opState_RewindMotorStarter  ; Rewind Motor output logical State
RSET SSR6_Rewind_Mtr_Starter  ; SSR6 Rewind Motor Run output
; rung 63
LDNOT opForceEnable_UpperToolVac  ; Upper tool vacuum output Force enable
OUT TR0
AND opState_UpperToolVac  ; Upper tool vacuum output logical State
SET V1A_Upper_Tool_Vac  ; V1A Upper Tool Vac On output
LD TR0
ANDNOT opState_UpperToolVac  ; Upper tool vacuum output logical State
RSET V1A_Upper_Tool_Vac  ; V1A Upper Tool Vac On output
; rung 64
LDNOT opForceEnable_UpperToolVentClose  ; Upper tool vent close output Force enable
OUT TR0
AND opState_UpperToolVentClose  ; Upper tool vent close output logical State
SET V1B_Upper_Tool_Vent_Close  ; V1B Upper Tool Vent Close output
LD TR0
ANDNOT opState_UpperToolVentClose  ; Upper tool vent close output logical State
RSET V1B_Upper_Tool_Vent_Close  ; V1B Upper Tool Vent Close output
; rung 65
LDNOT opForceEnable_LowerToolVac  ; Lower tool vacuum output Force enable
OUT TR0
AND opState_LowerToolVac  ; Lower tool vacuum output logical State
SET V2A_Lower_Tool_Vac  ; V2A Lower Tool Vacuum On output
LD TR0
ANDNOT opState_LowerToolVac  ; Lower tool vacuum output logical State
RSET V2A_Lower_Tool_Vac  ; V2A Lower Tool Vacuum On output

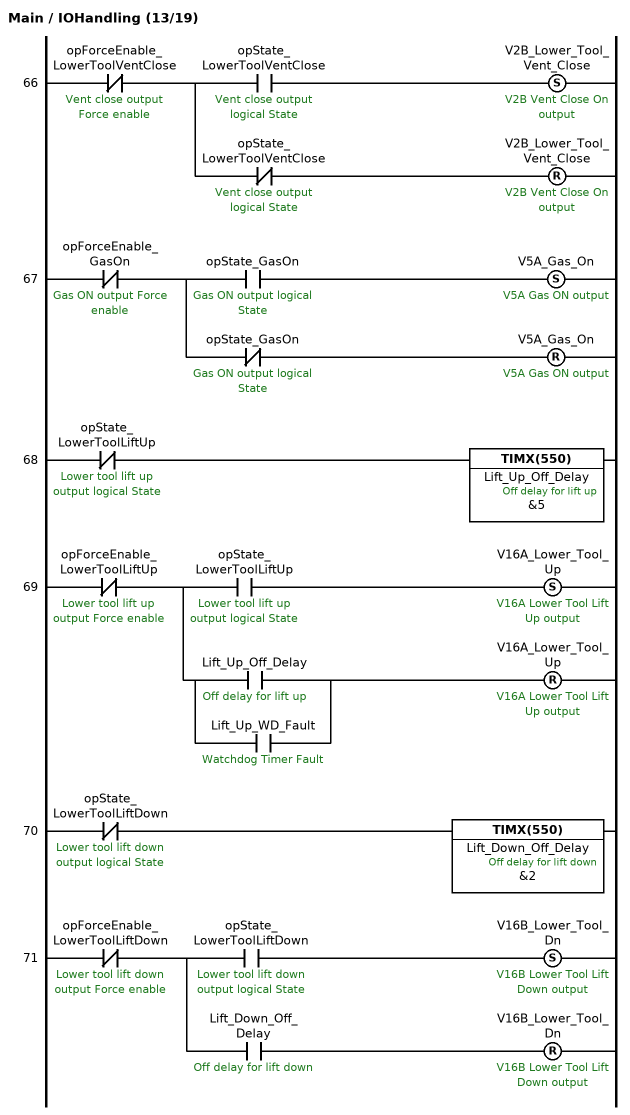
; rung 66
LDNOT opForceEnable_LowerToolVentClose  ; Vent close output Force enable
OUT TR0
AND opState_LowerToolVentClose  ; Vent close output logical State
SET V2B_Lower_Tool_Vent_Close  ; V2B Vent Close On output
LD TR0
ANDNOT opState_LowerToolVentClose  ; Vent close output logical State
RSET V2B_Lower_Tool_Vent_Close  ; V2B Vent Close On output
; rung 67
LDNOT opForceEnable_GasOn  ; Gas ON output Force enable
OUT TR0
AND opState_GasOn  ; Gas ON output logical State
SET V5A_Gas_On  ; V5A Gas ON output
LD TR0
ANDNOT opState_GasOn  ; Gas ON output logical State
RSET V5A_Gas_On  ; V5A Gas ON output
; rung 68
LDNOT opState_LowerToolLiftUp  ; Lower tool lift up output logical State
TIMX(550) Lift_Up_Off_Delay &5  ; Off delay for lift up
; rung 69
LDNOT opForceEnable_LowerToolLiftUp  ; Lower tool lift up output Force enable
OUT TR0
AND opState_LowerToolLiftUp  ; Lower tool lift up output logical State
SET V16A_Lower_Tool_Up  ; V16A Lower Tool Lift Up output
LD TR0
LD Lift_Up_Off_Delay  ; Off delay for lift up
OR Lift_Up_WD_Fault  ; Watchdog Timer Fault
ANDLD
RSET V16A_Lower_Tool_Up  ; V16A Lower Tool Lift Up output
; rung 70
LDNOT opState_LowerToolLiftDown  ; Lower tool lift down output logical State
TIMX(550) Lift_Down_Off_Delay &2  ; Off delay for lift down
; rung 71
LDNOT opForceEnable_LowerToolLiftDown  ; Lower tool lift down output Force enable
OUT TR0
AND opState_LowerToolLiftDown  ; Lower tool lift down output logical State
SET V16B_Lower_Tool_Dn  ; V16B Lower Tool Lift Down output
LD TR0
AND Lift_Down_Off_Delay  ; Off delay for lift down
RSET V16B_Lower_Tool_Dn  ; V16B Lower Tool Lift Down output

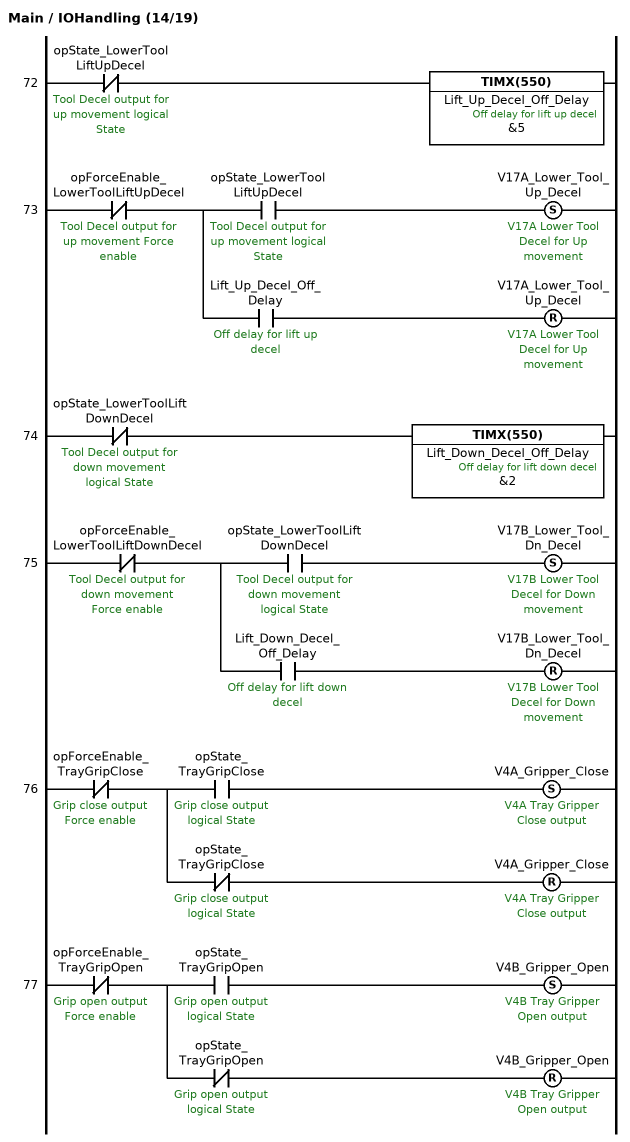
; rung 72
LDNOT opState_LowerToolLiftUpDecel  ; Tool Decel output for up movement logical State
TIMX(550) Lift_Up_Decel_Off_Delay &5  ; Off delay for lift up decel
; rung 73
LDNOT opForceEnable_LowerToolLiftUpDecel  ; Tool Decel output for up movement Force enable
OUT TR0
AND opState_LowerToolLiftUpDecel  ; Tool Decel output for up movement logical State
SET V17A_Lower_Tool_Up_Decel  ; V17A Lower Tool Decel for Up movement
LD TR0
AND Lift_Up_Decel_Off_Delay  ; Off delay for lift up decel
RSET V17A_Lower_Tool_Up_Decel  ; V17A Lower Tool Decel for Up movement
; rung 74
LDNOT opState_LowerToolLiftDownDecel  ; Tool Decel output for down movement logical State
TIMX(550) Lift_Down_Decel_Off_Delay &2  ; Off delay for lift down decel
; rung 75
LDNOT opForceEnable_LowerToolLiftDownDecel  ; Tool Decel output for down movement Force enable
OUT TR0
AND opState_LowerToolLiftDownDecel  ; Tool Decel output for down movement logical State
SET V17B_Lower_Tool_Dn_Decel  ; V17B Lower Tool Decel for Down movement
LD TR0
AND Lift_Down_Decel_Off_Delay  ; Off delay for lift down decel
RSET V17B_Lower_Tool_Dn_Decel  ; V17B Lower Tool Decel for Down movement
; rung 76
LDNOT opForceEnable_TrayGripClose  ; Grip close output Force enable
OUT TR0
AND opState_TrayGripClose  ; Grip close output logical State
SET V4A_Gripper_Close  ; V4A Tray Gripper Close output
LD TR0
ANDNOT opState_TrayGripClose  ; Grip close output logical State
RSET V4A_Gripper_Close  ; V4A Tray Gripper Close output
; rung 77
LDNOT opForceEnable_TrayGripOpen  ; Grip open output Force enable
OUT TR0
AND opState_TrayGripOpen  ; Grip open output logical State
SET V4B_Gripper_Open  ; V4B Tray Gripper Open output
LD TR0
ANDNOT opState_TrayGripOpen  ; Grip open output logical State
RSET V4B_Gripper_Open  ; V4B Tray Gripper Open output

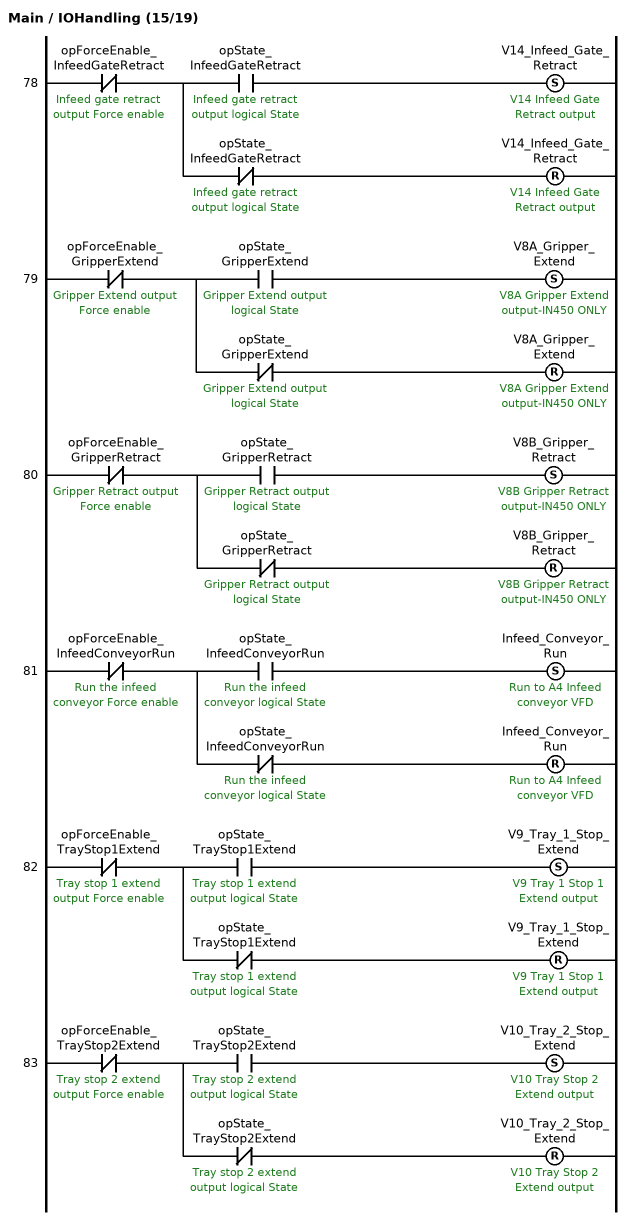
; rung 78
LDNOT opForceEnable_InfeedGateRetract  ; Infeed gate retract output Force enable
OUT TR0
AND opState_InfeedGateRetract  ; Infeed gate retract output logical State
SET V14_Infeed_Gate_Retract  ; V14 Infeed Gate Retract output
LD TR0
ANDNOT opState_InfeedGateRetract  ; Infeed gate retract output logical State
RSET V14_Infeed_Gate_Retract  ; V14 Infeed Gate Retract output
; rung 79
LDNOT opForceEnable_GripperExtend  ; Gripper Extend output Force enable
OUT TR0
AND opState_GripperExtend  ; Gripper Extend output logical State
SET V8A_Gripper_Extend  ; V8A Gripper Extend output-IN450 ONLY
LD TR0
ANDNOT opState_GripperExtend  ; Gripper Extend output logical State
RSET V8A_Gripper_Extend  ; V8A Gripper Extend output-IN450 ONLY
; rung 80
LDNOT opForceEnable_GripperRetract  ; Gripper Retract output Force enable
OUT TR0
AND opState_GripperRetract  ; Gripper Retract output logical State
SET V8B_Gripper_Retract  ; V8B Gripper Retract output-IN450 ONLY
LD TR0
ANDNOT opState_GripperRetract  ; Gripper Retract output logical State
RSET V8B_Gripper_Retract  ; V8B Gripper Retract output-IN450 ONLY
; rung 81
LDNOT opForceEnable_InfeedConveyorRun  ; Run the infeed conveyor Force enable
OUT TR0
AND opState_InfeedConveyorRun  ; Run the infeed conveyor logical State
SET Infeed_Conveyor_Run  ; Run to A4 Infeed conveyor VFD
LD TR0
ANDNOT opState_InfeedConveyorRun  ; Run the infeed conveyor logical State
RSET Infeed_Conveyor_Run  ; Run to A4 Infeed conveyor VFD
; rung 82
LDNOT opForceEnable_TrayStop1Extend  ; Tray stop 1 extend output Force enable
OUT TR0
AND opState_TrayStop1Extend  ; Tray stop 1 extend output logical State
SET V9_Tray_1_Stop_Extend  ; V9 Tray 1 Stop 1 Extend output
LD TR0
ANDNOT opState_TrayStop1Extend  ; Tray stop 1 extend output logical State
RSET V9_Tray_1_Stop_Extend  ; V9 Tray 1 Stop 1 Extend output
; rung 83
LDNOT opForceEnable_TrayStop2Extend  ; Tray stop 2 extend output Force enable
OUT TR0
AND opState_TrayStop2Extend  ; Tray stop 2 extend output logical State
SET V10_Tray_2_Stop_Extend  ; V10 Tray Stop 2 Extend output
LD TR0
ANDNOT opState_TrayStop2Extend  ; Tray stop 2 extend output logical State
RSET V10_Tray_2_Stop_Extend  ; V10 Tray Stop 2 Extend output

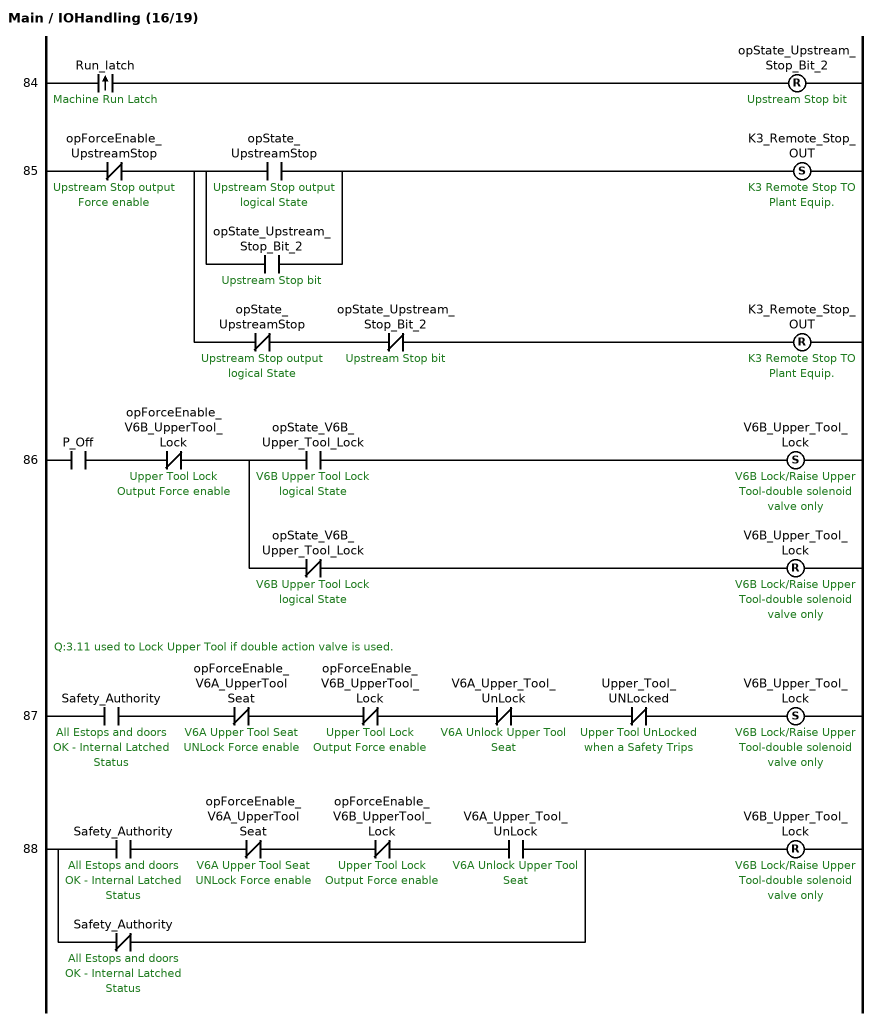
; rung 84
@LD Run_latch  ; Machine Run Latch
RSET opState_Upstream_Stop_Bit_2  ; Upstream Stop bit
; rung 85
LDNOT opForceEnable_UpstreamStop  ; Upstream Stop output Force enable
OUT TR0
LD opState_UpstreamStop  ; Upstream Stop output logical State
OR opState_Upstream_Stop_Bit_2  ; Upstream Stop bit
ANDLD
SET K3_Remote_Stop_OUT  ; K3 Remote Stop TO Plant Equip.
LD TR0
ANDNOT opState_UpstreamStop  ; Upstream Stop output logical State
ANDNOT opState_Upstream_Stop_Bit_2  ; Upstream Stop bit
RSET K3_Remote_Stop_OUT  ; K3 Remote Stop TO Plant Equip.
; rung 86
LD P_Off
ANDNOT opForceEnable_V6B_UpperTool_Lock  ; Upper Tool Lock Output Force enable
OUT TR0
AND opState_V6B_Upper_Tool_Lock  ; V6B Upper Tool Lock logical State
SET V6B_Upper_Tool_Lock  ; V6B Lock/Raise Upper Tool-double solenoid valve only
LD TR0
ANDNOT opState_V6B_Upper_Tool_Lock  ; V6B Upper Tool Lock logical State
RSET V6B_Upper_Tool_Lock  ; V6B Lock/Raise Upper Tool-double solenoid valve only
; rung 87: Q:3.11 used to Lock Upper Tool if double action valve is used.
LD Safety_Authority  ; All Estops and doors OK - Internal Latched Status
ANDNOT opForceEnable_V6A_UpperToolSeat  ; V6A Upper Tool Seat UNLock Force enable
ANDNOT opForceEnable_V6B_UpperTool_Lock  ; Upper Tool Lock Output Force enable
ANDNOT V6A_Upper_Tool_UnLock  ; V6A Unlock Upper Tool Seat
ANDNOT Upper_Tool_UNLocked  ; Upper Tool UnLocked when a Safety Trips
SET V6B_Upper_Tool_Lock  ; V6B Lock/Raise Upper Tool-double solenoid valve only
; rung 88
LD Safety_Authority  ; All Estops and doors OK - Internal Latched Status
ANDNOT opForceEnable_V6A_UpperToolSeat  ; V6A Upper Tool Seat UNLock Force enable
ANDNOT opForceEnable_V6B_UpperTool_Lock  ; Upper Tool Lock Output Force enable
AND V6A_Upper_Tool_UnLock  ; V6A Unlock Upper Tool Seat
ORNOT Safety_Authority  ; All Estops and doors OK - Internal Latched Status
RSET V6B_Upper_Tool_Lock  ; V6B Lock/Raise Upper Tool-double solenoid valve only

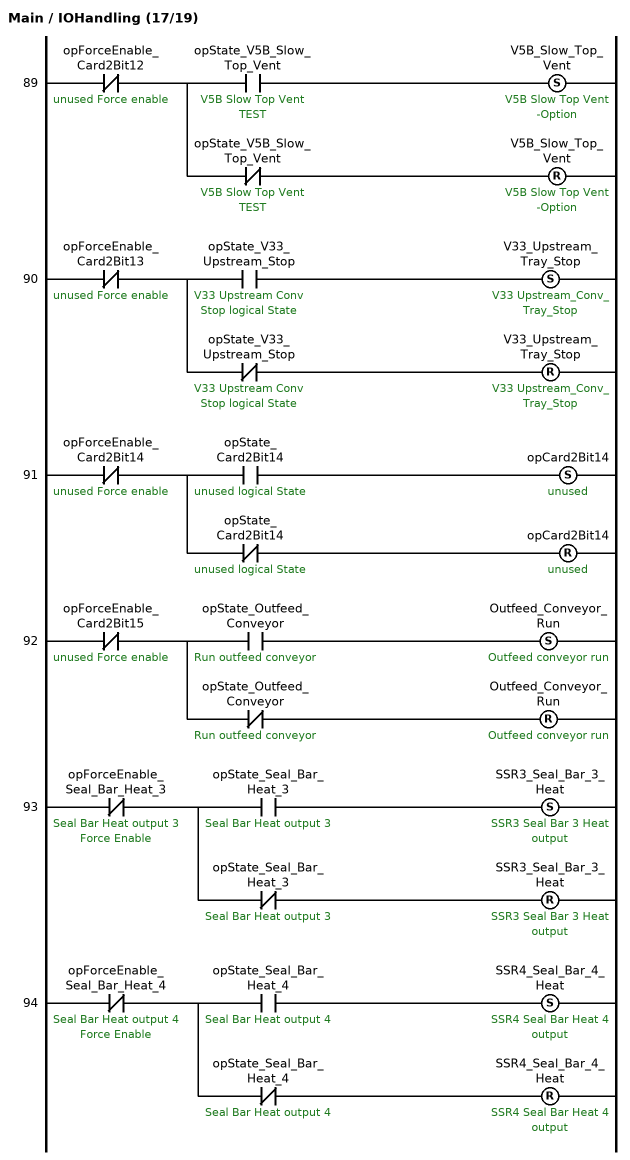
; rung 89
LDNOT opForceEnable_Card2Bit12  ; unused Force enable
OUT TR0
AND opState_V5B_Slow_Top_Vent  ; V5B Slow Top Vent TEST
SET V5B_Slow_Top_Vent  ; V5B Slow Top Vent -Option
LD TR0
ANDNOT opState_V5B_Slow_Top_Vent  ; V5B Slow Top Vent TEST
RSET V5B_Slow_Top_Vent  ; V5B Slow Top Vent -Option
; rung 90
LDNOT opForceEnable_Card2Bit13  ; unused Force enable
OUT TR0
AND opState_V33_Upstream_Stop  ; V33 Upstream Conv Stop logical State
SET V33_Upstream_Tray_Stop  ; V33 Upstream_Conv_Tray_Stop
LD TR0
ANDNOT opState_V33_Upstream_Stop  ; V33 Upstream Conv Stop logical State
RSET V33_Upstream_Tray_Stop  ; V33 Upstream_Conv_Tray_Stop
; rung 91
LDNOT opForceEnable_Card2Bit14  ; unused Force enable
OUT TR0
AND opState_Card2Bit14  ; unused logical State
SET opCard2Bit14  ; unused
LD TR0
ANDNOT opState_Card2Bit14  ; unused logical State
RSET opCard2Bit14  ; unused
; rung 92
LDNOT opForceEnable_Card2Bit15  ; unused Force enable
OUT TR0
AND opState_Outfeed_Conveyor  ; Run outfeed conveyor
SET Outfeed_Conveyor_Run  ; Outfeed conveyor run
LD TR0
ANDNOT opState_Outfeed_Conveyor  ; Run outfeed conveyor
RSET Outfeed_Conveyor_Run  ; Outfeed conveyor run
; rung 93
LDNOT opForceEnable_Seal_Bar_Heat_3  ; Seal Bar Heat output 3 Force Enable
OUT TR0
AND opState_Seal_Bar_Heat_3  ; Seal Bar Heat output 3
SET SSR3_Seal_Bar_3_Heat  ; SSR3 Seal Bar 3 Heat output
LD TR0
ANDNOT opState_Seal_Bar_Heat_3  ; Seal Bar Heat output 3
RSET SSR3_Seal_Bar_3_Heat  ; SSR3 Seal Bar 3 Heat output
; rung 94
LDNOT opForceEnable_Seal_Bar_Heat_4  ; Seal Bar Heat output 4 Force Enable
OUT TR0
AND opState_Seal_Bar_Heat_4  ; Seal Bar Heat output 4
SET SSR4_Seal_Bar_4_Heat  ; SSR4 Seal Bar Heat 4 output
LD TR0
ANDNOT opState_Seal_Bar_Heat_4  ; Seal Bar Heat output 4
RSET SSR4_Seal_Bar_4_Heat  ; SSR4 Seal Bar Heat 4 output

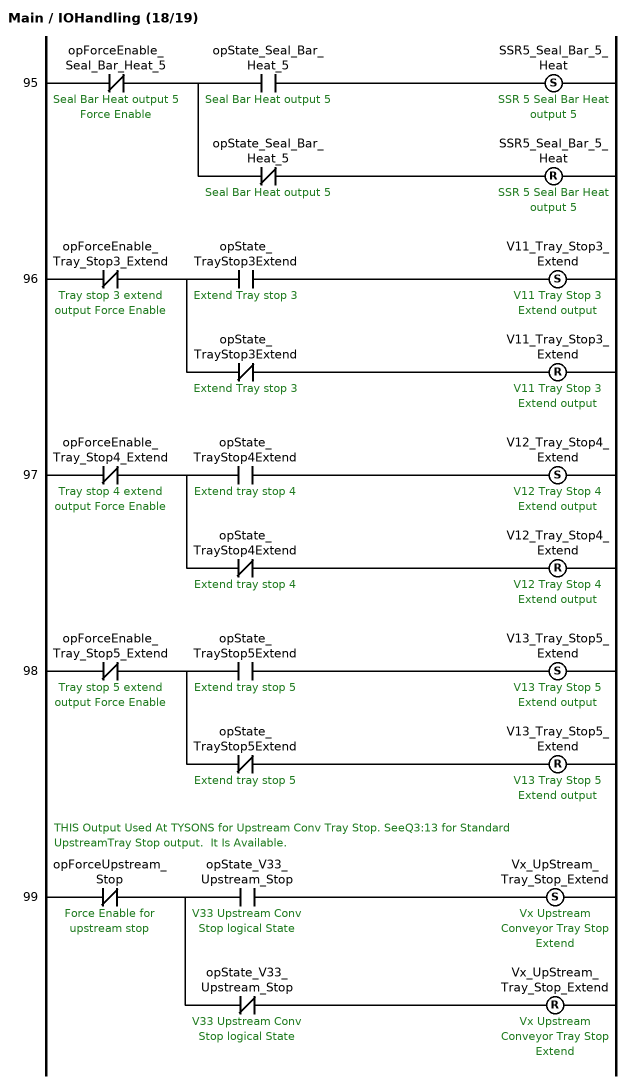
; rung 95
LDNOT opForceEnable_Seal_Bar_Heat_5  ; Seal Bar Heat output 5 Force Enable
OUT TR0
AND opState_Seal_Bar_Heat_5  ; Seal Bar Heat output 5
SET SSR5_Seal_Bar_5_Heat  ; SSR 5 Seal Bar Heat output 5
LD TR0
ANDNOT opState_Seal_Bar_Heat_5  ; Seal Bar Heat output 5
RSET SSR5_Seal_Bar_5_Heat  ; SSR 5 Seal Bar Heat output 5
; rung 96
LDNOT opForceEnable_Tray_Stop3_Extend  ; Tray stop 3 extend output Force Enable
OUT TR0
AND opState_TrayStop3Extend  ; Extend Tray stop 3
SET V11_Tray_Stop3_Extend  ; V11 Tray Stop 3 Extend output
LD TR0
ANDNOT opState_TrayStop3Extend  ; Extend Tray stop 3
RSET V11_Tray_Stop3_Extend  ; V11 Tray Stop 3 Extend output
; rung 97
LDNOT opForceEnable_Tray_Stop4_Extend  ; Tray stop 4 extend output Force Enable
OUT TR0
AND opState_TrayStop4Extend  ; Extend tray stop 4
SET V12_Tray_Stop4_Extend  ; V12 Tray Stop 4 Extend output
LD TR0
ANDNOT opState_TrayStop4Extend  ; Extend tray stop 4
RSET V12_Tray_Stop4_Extend  ; V12 Tray Stop 4 Extend output
; rung 98
LDNOT opForceEnable_Tray_Stop5_Extend  ; Tray stop 5 extend output Force Enable
OUT TR0
AND opState_TrayStop5Extend  ; Extend tray stop 5
SET V13_Tray_Stop5_Extend  ; V13 Tray Stop 5 Extend output
LD TR0
ANDNOT opState_TrayStop5Extend  ; Extend tray stop 5
RSET V13_Tray_Stop5_Extend  ; V13 Tray Stop 5 Extend output
; rung 99: THIS Output Used At TYSONS for Upstream Conv Tray Stop. SeeQ3:13 for Standard UpstreamTray Stop output.  It Is Available.
LDNOT opForceUpstream_Stop  ; Force Enable for upstream stop
OUT TR0
AND opState_V33_Upstream_Stop  ; V33 Upstream Conv Stop logical State
SET Vx_UpStream_Tray_Stop_Extend  ; Vx Upstream Conveyor Tray Stop Extend
LD TR0
ANDNOT opState_V33_Upstream_Stop  ; V33 Upstream Conv Stop logical State
RSET Vx_UpStream_Tray_Stop_Extend  ; Vx Upstream Conveyor Tray Stop Extend

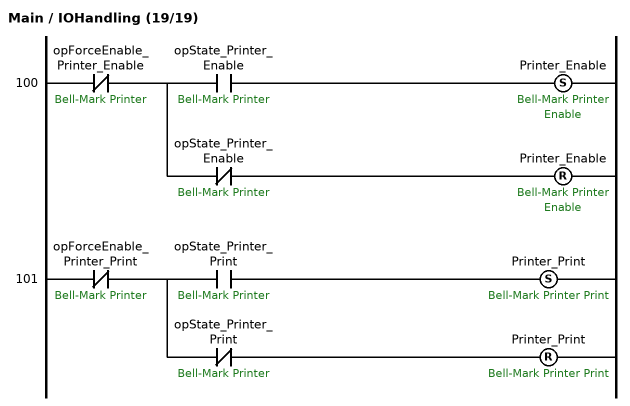
; rung 100
LDNOT opForceEnable_Printer_Enable  ; Bell-Mark Printer
OUT TR0
AND opState_Printer_Enable  ; Bell-Mark Printer
SET Printer_Enable  ; Bell-Mark Printer Enable
LD TR0
ANDNOT opState_Printer_Enable  ; Bell-Mark Printer
RSET Printer_Enable  ; Bell-Mark Printer Enable
; rung 101
LDNOT opForceEnable_Printer_Print  ; Bell-Mark Printer
OUT TR0
AND opState_Printer_Print  ; Bell-Mark Printer
SET Printer_Print  ; Bell-Mark Printer Print
LD TR0
ANDNOT opState_Printer_Print  ; Bell-Mark Printer
RSET Printer_Print  ; Bell-Mark Printer Print

### Section Gripper_Jog_Sequence

